FUNCTION_BLOCK AD_TO_AR_NUM (* Composite FB for numerically converting AD (DWORD) adapter to AR (REAL) adapter (via UDINT, not a bit-reinterpretation) *)
  (* Standard: 61499-2; Description: Copyright (c) 2026 HR Agrartechnik GmbH This program and the accompanying materials are made available under the terms of the Eclipse Public License 2.0 which is available at https://www.eclipse.org/legal/epl-2.0/ SPDX-License-Identifier: EPL-2.0 *)
  (* Version 1.0, 2026-08-30, Franz Höpfinger, HR Agrartechnik GmbH *)
  PACKAGE adapter::conversion::unidirectional;
  (* Documentation:
  AD_TO_AR_NUM
   🇩🇪 Deutsch
   Numerisch korrekte Alternative zu AD_TO_AR. Wandelt einen DWORD-Adapter (AD_IN) über einen internen UDINT-Zwischenschritt in einen REAL-Adapter (AR_OUT) um — echte Wertumwandlung, keine Bit-Reinterpretation.
   Warum nicht einfach AD_TO_AR?
   AD_TO_AR nutzt intern F_DWORD_TO_REAL, was im FORTE-Kern für Bit-String-Typen (DWORD/WORD/BYTE/LWORD) eine reine IEEE754-Bit-Reinterpretation ist, keinen numerischen Cast. Ein roher Zähler-/Analogwert wie DWORD#2048 würde dadurch NICHT zu REAL#2048.0, sondern zu einer bedeutungslosen Zahl nahe Null.
   AD_TO_AR_NUM vermeidet diese Falle, indem es zweistufig über F_DWORD_TO_UDINT (Bit-Reinterpretation DWORD→UDINT, hier gültig, da beide dieselbe 32-bit-Darstellung eines vorzeichenlosen Integers teilen) und anschließend F_UDINT_TO_REAL (echter numerischer Cast) konvertiert — dieselbe Kette, die bereits in mehreren Übungen (Uebung_028a_AR u.a.) von Hand verdrahtet wird, hier als ein einziger, drop-in-kompatibler Baustein.
   Wann welchen Baustein verwenden?
    - AD_TO_AR_NUM: Der DWORD-Wert ist eine Zahl (z. B. Analog-Rohwert, Zähler) und soll als derselbe Zahlenwert in REAL vorliegen.
   - AD_TO_AR: Der DWORD-Wert ist bereits ein Bitmuster, das als REAL interpretiert werden soll (z. B. Ergebnis von F_REAL_TO_DWORD, seriellisierte Float-Daten).
    🇬🇧 English
   Numerically correct alternative to AD_TO_AR. Converts a DWORD adapter (AD_IN) into a REAL adapter (AR_OUT) via an internal UDINT step — a real value conversion, not a bit-reinterpretation.
   Why not just use AD_TO_AR?
   AD_TO_AR internally uses F_DWORD_TO_REAL, which in the FORTE core is a pure IEEE754 bit-reinterpretation for bit-string types (DWORD/WORD/BYTE/LWORD), not a numeric cast. A raw counter/analog value such as DWORD#2048 would NOT become REAL#2048.0 but a meaningless value near zero.
   AD_TO_AR_NUM avoids this trap by converting in two steps via F_DWORD_TO_UDINT (bit-reinterpretation DWORD→UDINT, valid here since both share the same 32-bit unsigned-integer representation) and then F_UDINT_TO_REAL (a real numeric cast) — the same chain already wired by hand in several exercises (Uebung_028a_AR and others), packaged here as a single drop-in-compatible block.
   Which block to use?
    - AD_TO_AR_NUM: The DWORD value is a number (e.g. raw analog value, counter) and should carry the same numeric value as REAL.
   - AD_TO_AR: The DWORD value is already a bit pattern meant to be interpreted as REAL (e.g. the result of F_REAL_TO_DWORD, serialized float data).
  *)
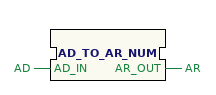
  SOCKETS
    AD_IN : adapter::types::unidirectional::AD; (* DWORD Adapter Input *)
  END_SOCKETS
  PLUGS
    AR_OUT : adapter::types::unidirectional::AR; (* REAL Adapter Output *)
  END_PLUGS
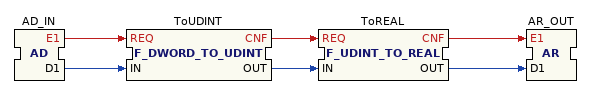
  FBS
    ToUDINT : iec61131::conversion::F_DWORD_TO_UDINT;
    ToREAL : iec61131::conversion::F_UDINT_TO_REAL;
  END_FBS
  EVENT_CONNECTIONS
    AD_IN.E1 TO ToUDINT.REQ;
    ToUDINT.CNF TO ToREAL.REQ;
    ToREAL.CNF TO AR_OUT.E1;
  END_CONNECTIONS
  DATA_CONNECTIONS
    AD_IN.D1 TO ToUDINT.IN;
    ToUDINT.OUT TO ToREAL.IN;
    ToREAL.OUT TO AR_OUT.D1;
  END_CONNECTIONS
END_FUNCTION_BLOCK
